// TIA Portal V20 export
FUNCTION_BLOCK "LER_RFID_Mobile"   // FB191, LAD
// stored: Access Published, MemoryReserve 100, SetENOAutomatically false
   VAR_INPUT
      enable : Bool;
      enableManualCmds : Bool;
   END_VAR
   VAR_OUTPUT
      error : Bool;
      status : DWord;
   END_VAR
   VAR_IN_OUT
      IdentRfAntena : "LSicar_typeIdentInterfaceHmi";
      moduleInterface : "LER_typeMobileRFIDInterface";
   END_VAR
   VAR
      instTRCV_C : TRCV_C;
      statConnectionData : TCON_IP_v4;
      statTrcvUDT : "LER_typeTrcvUDT";
      statResultRFIDReset : Bool;
      statPulse : Array[0..9] of Bool;
      statTonTimer : TON_TIME;
      statBobinData : IID_IN_I_81;
      statRFID_str : String[32];
      statEPCID_str : String[32];
      statHi : Byte;
      statLo : Byte;
      statHexArray : Array[0..15] of Char;
   END_VAR
   VAR_TEMP
      resultRFID_Delete : String;
      resultData_Delete : WString;
      resultid_Delete : SInt;
      tempRet_Val : Word;
      tempBobinEPCData : Array[1..62] of Byte;
      i : Int;
      HI : Int;
      LO : Int;
   END_VAR
   VAR CONSTANT
      TRUE : Bool := true;
      FALSE : Bool;
      deviceType : WString := WSTRING#'RF160B';
      deviceId : SInt := 1;   // RF600 = 6, RF100 = 1
      tagType : WString := WSTRING#'RFID';
   END_VAR
   // statHexArray[0] := '0';
   // statHexArray[1] := '1';
   // statHexArray[2] := '2';
   // statHexArray[3] := '3';
   // statHexArray[4] := '4';
   // statHexArray[5] := '5';
   // statHexArray[6] := '6';
   // statHexArray[7] := '7';
   // statHexArray[8] := '8';
   // statHexArray[9] := '9';
   // statHexArray[10] := 'A';
   // statHexArray[11] := 'B';
   // statHexArray[12] := 'C';
   // statHexArray[13] := 'D';
   // statHexArray[14] := 'E';
   // statHexArray[15] := 'F';
BEGIN

REGION Network 1 (SCL): Input Mapping
   // TRCV_C
   #statTrcvUDT.Input.Enable := #TRUE;
   #statTrcvUDT.Input.Len := 0;
   #statTrcvUDT.Input.Adhoc := #TRUE;
   //#statTrcvUDT.InOut.ADDR := #FALSE;
   //#statTrcvUDT.InOut.COM_RST := #FALSE;

   // TCON_IP V4
   #statConnectionData.InterfaceId := 120;
   #statConnectionData.ID := 16#0001;
   #statConnectionData.LocalPort := 2000;

   // Manual Commands
   IF #enableManualCmds OR true THEN
       #statTrcvUDT.Input.Cont := NOT #moduleInterface.commands.ResetReq AND NOT #IdentRfAntena.pushbutton.%X0;
       #statResultRFIDReset := #moduleInterface.commands.resultRFIDReset OR #IdentRfAntena.pushbutton.%X3;
   END_IF;
END_REGION

REGION Network 2: TRCV
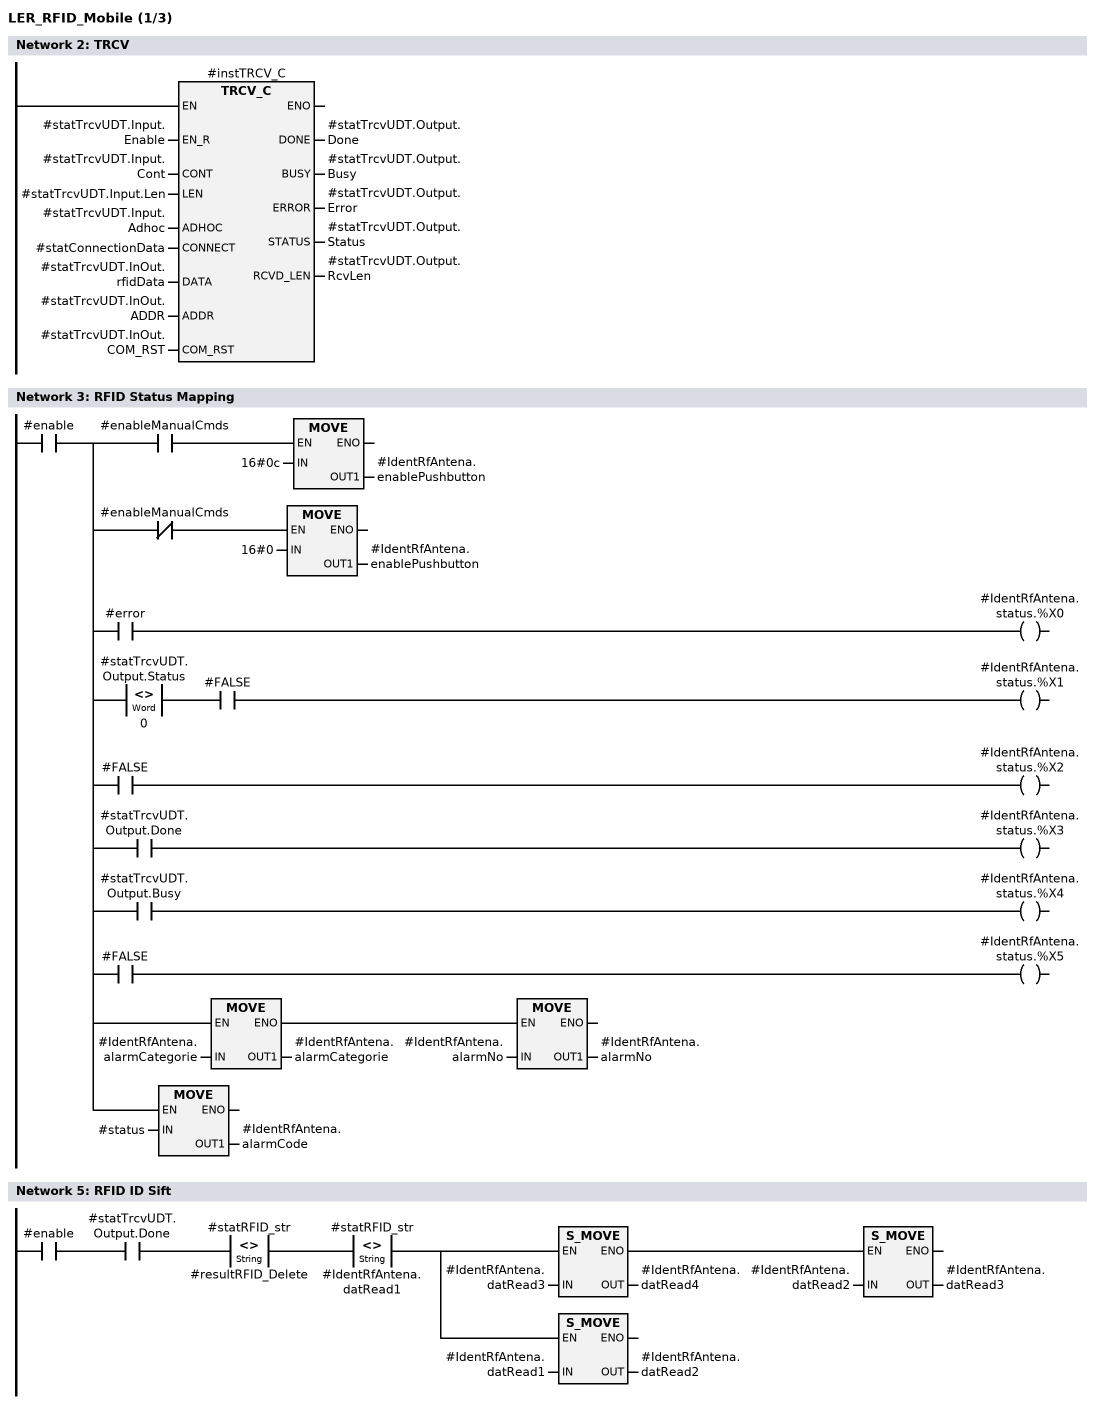
   RUNG wire#powerrail
      #instTRCV_C.TRCV_C(EN_R := #statTrcvUDT.Input.Enable, CONT := #statTrcvUDT.Input.Cont, LEN := #statTrcvUDT.Input.Len, ADHOC := #statTrcvUDT.Input.Adhoc, CONNECT := #statConnectionData, DATA := #statTrcvUDT.InOut.rfidData, ADDR := #statTrcvUDT.InOut.ADDR, COM_RST := #statTrcvUDT.InOut.COM_RST, DONE => #statTrcvUDT.Output.Done, BUSY => #statTrcvUDT.Output.Busy, ERROR => #statTrcvUDT.Output.Error, STATUS => #statTrcvUDT.Output.Status, RCVD_LEN => #statTrcvUDT.Output.RcvLen)
   END_RUNG
   // the same network as SCL:
   #instTRCV_C(EN_R := #statTrcvUDT.Input.Enable,   // TRCV_C
               CONT := #statTrcvUDT.Input.Cont,
               LEN := #statTrcvUDT.Input.Len,
               ADHOC := #statTrcvUDT.Input.Adhoc,
               CONNECT := #statConnectionData,
               DATA := #statTrcvUDT.InOut.rfidData,
               ADDR := #statTrcvUDT.InOut.ADDR,
               COM_RST := #statTrcvUDT.InOut.COM_RST,
               DONE => #statTrcvUDT.Output.Done,
               BUSY => #statTrcvUDT.Output.Busy,
               ERROR => #statTrcvUDT.Output.Error,
               STATUS => #statTrcvUDT.Output.Status,
               RCVD_LEN => #statTrcvUDT.Output.RcvLen);
END_REGION

REGION Network 3: RFID Status Mapping
   RUNG wire#powerrail
      Contact( #enable )
      wire#w1
      Contact( #enableManualCmds )
      Move(in := 16#0c, out1 => #IdentRfAntena.enablePushbutton)
   END_RUNG
   RUNG wire#w1
      I_Contact( #enableManualCmds )
      Move(in := 16#0, out1 => #IdentRfAntena.enablePushbutton)
   END_RUNG
   RUNG wire#w1
      Contact( #error )
      Coil( #IdentRfAntena.status.%X0 )
   END_RUNG
   RUNG wire#w1
      { S7_Templates := "SrcType := Word" } NE_Contact(in1 := #statTrcvUDT.Output.Status, in2 := 0)
      Contact( #FALSE )
      Coil( #IdentRfAntena.status.%X1 )
   END_RUNG
   RUNG wire#w1
      Contact( #FALSE )
      Coil( #IdentRfAntena.status.%X2 )
   END_RUNG
   RUNG wire#w1
      Contact( #statTrcvUDT.Output.Done )
      Coil( #IdentRfAntena.status.%X3 )
   END_RUNG
   RUNG wire#w1
      Contact( #statTrcvUDT.Output.Busy )
      Coil( #IdentRfAntena.status.%X4 )
   END_RUNG
   RUNG wire#w1
      Contact( #FALSE )
      Coil( #IdentRfAntena.status.%X5 )
   END_RUNG
   RUNG wire#w1
      Move(in := #IdentRfAntena.alarmCategorie, out1 => #IdentRfAntena.alarmCategorie)
      Move(in := #IdentRfAntena.alarmNo, out1 => #IdentRfAntena.alarmNo)
   END_RUNG
   RUNG wire#w1
      Move(in := #status, out1 => #IdentRfAntena.alarmCode)
   END_RUNG
   // the same network as SCL:
   IF #enable AND #enableManualCmds THEN #IdentRfAntena.enablePushbutton := 16#0c; END_IF;
   IF #enable AND NOT #enableManualCmds THEN #IdentRfAntena.enablePushbutton := 16#0; END_IF;
   #IdentRfAntena.status.%X0 := #enable AND #error;
   #IdentRfAntena.status.%X1 := #enable AND (#statTrcvUDT.Output.Status <> 0) AND #FALSE;
   #IdentRfAntena.status.%X2 := #enable AND #FALSE;
   #IdentRfAntena.status.%X3 := #enable AND #statTrcvUDT.Output.Done;
   #IdentRfAntena.status.%X4 := #enable AND #statTrcvUDT.Output.Busy;
   #IdentRfAntena.status.%X5 := #enable AND #FALSE;
   IF #enable THEN
       #IdentRfAntena.alarmCategorie := #IdentRfAntena.alarmCategorie;
       #IdentRfAntena.alarmNo := #IdentRfAntena.alarmNo;
       #IdentRfAntena.alarmCode := #status;
   END_IF;
END_REGION

REGION Network 4 (SCL): RFID combination (Byte To string)
   IF #enable AND #statTrcvUDT.Output.Done THEN
       #statRFID_str := '';

       FOR #i := 0 TO 15 DO
           #statHi := SHR(IN := #statTrcvUDT.InOut.rfidData[#i], N := 4);
           #statLo := #statTrcvUDT.InOut.rfidData[#i] AND 16#0F;
           #statRFID_str := CONCAT(IN1 := #statRFID_str, IN2 := #statHexArray[#statHi]);
           #statRFID_str := CONCAT(IN1 := #statRFID_str, IN2 := #statHexArray[#statLo]);
       END_FOR;
   END_IF;
END_REGION

REGION Network 5: RFID ID Sift
   RUNG wire#powerrail
      Contact( #enable )
      Contact( #statTrcvUDT.Output.Done )
      { S7_Templates := "SrcType := String" } NE_Contact(in1 := #statRFID_str, in2 := #resultRFID_Delete)
      { S7_Templates := "SrcType := String" } NE_Contact(in1 := #statRFID_str, in2 := #IdentRfAntena.datRead1)
      wire#w1
      S_Move(in := #IdentRfAntena.datRead3, out => #IdentRfAntena.datRead4)
      S_Move(in := #IdentRfAntena.datRead2, out => #IdentRfAntena.datRead3)
   END_RUNG
   RUNG wire#w1
      S_Move(in := #IdentRfAntena.datRead1, out => #IdentRfAntena.datRead2)
   END_RUNG
   // the same network as SCL:
   IF #enable AND #statTrcvUDT.Output.Done AND (#statRFID_str <> #resultRFID_Delete) AND (#statRFID_str <> #IdentRfAntena.datRead1) THEN
       #IdentRfAntena.datRead4 := #IdentRfAntena.datRead3;
       #IdentRfAntena.datRead3 := #IdentRfAntena.datRead2;
       #IdentRfAntena.datRead2 := #IdentRfAntena.datRead1;
   END_IF;
END_REGION

REGION Network 6: RFID ID Mapping
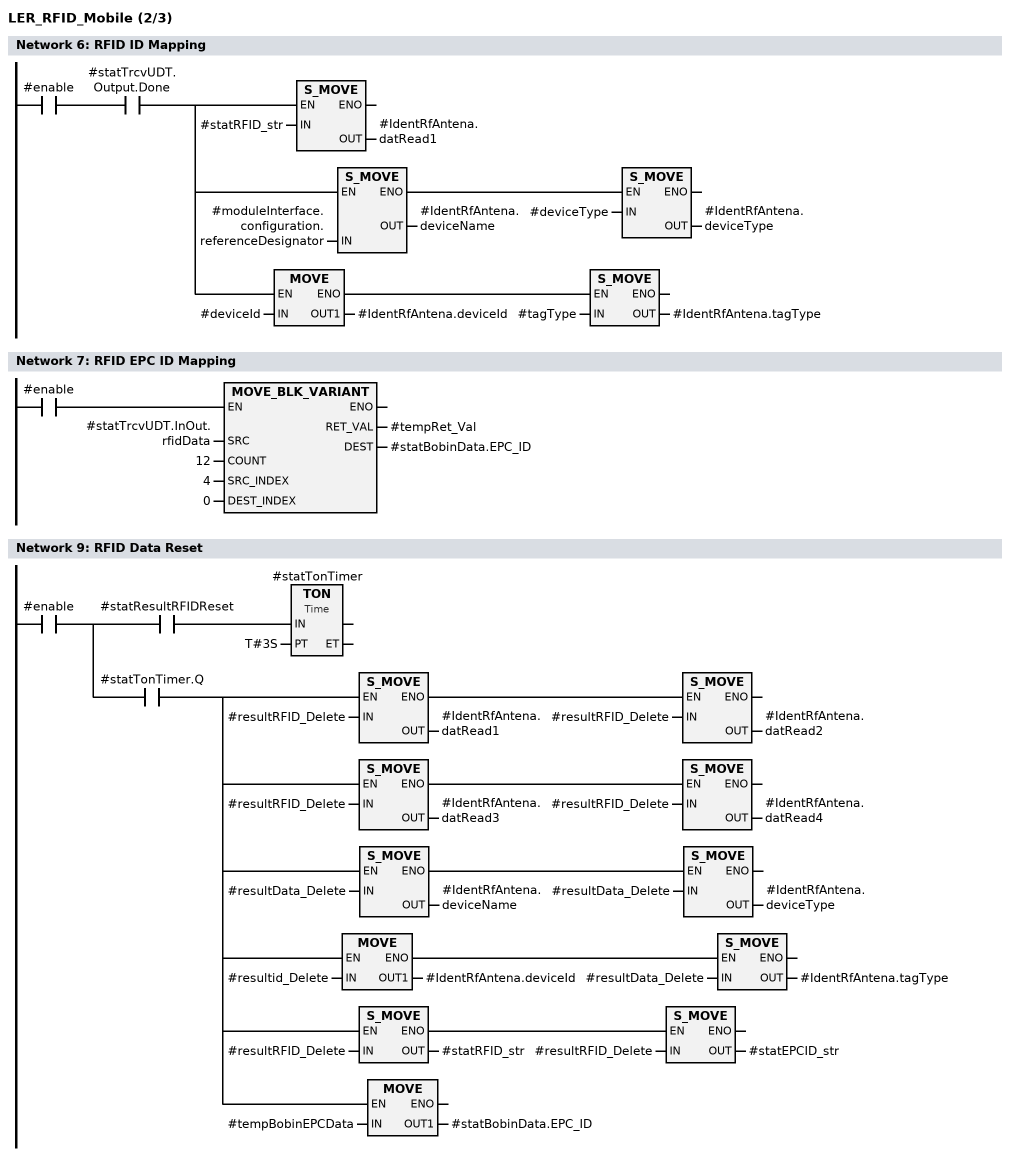
   RUNG wire#powerrail
      Contact( #enable )
      Contact( #statTrcvUDT.Output.Done )
      wire#w1
      S_Move(in := #statRFID_str, out => #IdentRfAntena.datRead1)
   END_RUNG
   RUNG wire#w1
      S_Move(in := #moduleInterface.configuration.referenceDesignator, out => #IdentRfAntena.deviceName)
      S_Move(in := #deviceType, out => #IdentRfAntena.deviceType)
   END_RUNG
   RUNG wire#w1
      Move(in := #deviceId, out1 => #IdentRfAntena.deviceId)
      S_Move(in := #tagType, out => #IdentRfAntena.tagType)
   END_RUNG
   // the same network as SCL:
   IF #enable AND #statTrcvUDT.Output.Done THEN
       #IdentRfAntena.datRead1 := #statRFID_str;
       #IdentRfAntena.deviceName := #moduleInterface.configuration.referenceDesignator;
       #IdentRfAntena.deviceType := #deviceType;
       #IdentRfAntena.deviceId := #deviceId;
       #IdentRfAntena.tagType := #tagType;
   END_IF;
END_REGION

REGION Network 7: RFID EPC ID Mapping
   RUNG wire#powerrail
      Contact( #enable )
      MOVE_BLK_VARIANT(SRC := #statTrcvUDT.InOut.rfidData, COUNT := 12, SRC_INDEX := 4, DEST_INDEX := 0, Ret_Val => #tempRet_Val, DEST => #statBobinData.EPC_ID)
   END_RUNG
   // the same network as SCL:
   IF #enable THEN
       #tempRet_Val := MOVE_BLK_VARIANT(SRC := #statTrcvUDT.InOut.rfidData,
                               COUNT := 12,
                               SRC_INDEX := 4,
                               DEST_INDEX := 0,
                               DEST => #statBobinData.EPC_ID);
   END_IF;
END_REGION

REGION Network 8 (SCL): RFID EPC ID Combination (Byte To string)
   IF #enable AND #statTrcvUDT.Output.Done THEN
       #statEPCID_str := '';

       FOR #i := 1 TO 12 DO
           #statHi := SHR(IN := #statBobinData.EPC_ID[#i], N := 4);
           #statLo := #statBobinData.EPC_ID[#i] AND 16#0F;
           #statEPCID_str := CONCAT(IN1 := #statEPCID_str, IN2 := #statHexArray[#statHi]);
           #statEPCID_str := CONCAT(IN1 := #statEPCID_str, IN2 := #statHexArray[#statLo]);
       END_FOR;
   END_IF;
END_REGION

REGION Network 9: RFID Data Reset
   RUNG wire#powerrail
      Contact( #enable )
      wire#w1
      Contact( #statResultRFIDReset )
      { S7_Templates := "time_type := Time" } #statTonTimer.TON(pt := T#3S, et =>)
   END_RUNG
   RUNG wire#w1
      Contact( #statTonTimer.Q )
      wire#w2
      S_Move(in := #resultRFID_Delete, out => #IdentRfAntena.datRead1)
      S_Move(in := #resultRFID_Delete, out => #IdentRfAntena.datRead2)
   END_RUNG
   RUNG wire#w2
      S_Move(in := #resultRFID_Delete, out => #IdentRfAntena.datRead3)
      S_Move(in := #resultRFID_Delete, out => #IdentRfAntena.datRead4)
   END_RUNG
   RUNG wire#w2
      S_Move(in := #resultData_Delete, out => #IdentRfAntena.deviceName)
      S_Move(in := #resultData_Delete, out => #IdentRfAntena.deviceType)
   END_RUNG
   RUNG wire#w2
      Move(in := #resultid_Delete, out1 => #IdentRfAntena.deviceId)
      S_Move(in := #resultData_Delete, out => #IdentRfAntena.tagType)
   END_RUNG
   RUNG wire#w2
      S_Move(in := #resultRFID_Delete, out => #statRFID_str)
      S_Move(in := #resultRFID_Delete, out => #statEPCID_str)
   END_RUNG
   RUNG wire#w2
      Move(in := #tempBobinEPCData, out1 => #statBobinData.EPC_ID)
   END_RUNG
   // the same network as SCL:
   #statTonTimer(IN := #enable AND #statResultRFIDReset, PT := T#3S);   // TON
   IF #enable AND #statTonTimer.Q THEN
       #IdentRfAntena.datRead1 := #resultRFID_Delete;
       #IdentRfAntena.datRead2 := #resultRFID_Delete;
       #IdentRfAntena.datRead3 := #resultRFID_Delete;
       #IdentRfAntena.datRead4 := #resultRFID_Delete;
       #IdentRfAntena.deviceName := #resultData_Delete;
       #IdentRfAntena.deviceType := #resultData_Delete;
       #IdentRfAntena.deviceId := #resultid_Delete;
       #IdentRfAntena.tagType := #resultData_Delete;
       #statRFID_str := #resultRFID_Delete;
       #statEPCID_str := #resultRFID_Delete;
       #statBobinData.EPC_ID := #tempBobinEPCData;
   END_IF;
END_REGION

REGION Network 10: Error Check
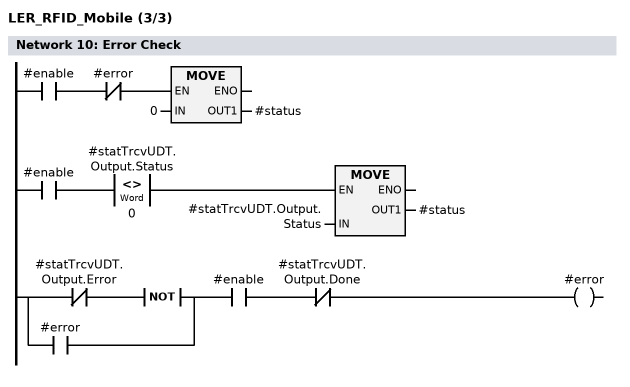
   RUNG wire#powerrail
      Contact( #enable )
      I_Contact( #error )
      Move(in := 0, out1 => #status)
   END_RUNG
   RUNG wire#powerrail
      Contact( #enable )
      { S7_Templates := "SrcType := Word" } NE_Contact(in1 := #statTrcvUDT.Output.Status, in2 := 0)
      Move(in := #statTrcvUDT.Output.Status, out1 => #status)
   END_RUNG
   RUNG wire#powerrail
      I_Contact( #statTrcvUDT.Output.Error )
      Not()
      wire#w1
      Contact( #enable )
      I_Contact( #statTrcvUDT.Output.Done )
      Coil( #error )
   END_RUNG
   RUNG wire#powerrail
      Contact( #error )
   END_RUNG wire#w1
   // the same network as SCL:
   IF #enable AND NOT #error THEN #status := 0; END_IF;
   IF #enable AND (#statTrcvUDT.Output.Status <> 0) THEN #status := #statTrcvUDT.Output.Status; END_IF;
   #error := (NOT (NOT #statTrcvUDT.Output.Error) OR #error) AND #enable AND NOT #statTrcvUDT.Output.Done;
END_REGION

REGION Network 11 (SCL): Output Mapping
   #moduleInterface.monitoring.ResultData := #IdentRfAntena;
   #moduleInterface.monitoring.error := #error;
   #moduleInterface.monitoring.status:= #status;
END_REGION
END_FUNCTION_BLOCK
